// TIA Portal project "ElectricShipPLC" (V17)

(* hardware
DEVICE "S7-1200 station_2"  S7-1200 Station
   slot 0: "Rack_0"  S7-1200 Rack  Rack  V1.0
   slot 1: "PLC_3"  CPU 1214C DC/DC/DC  6ES7 214-1AG40-0XB0  V4.5
*)

// ===== PLC "PLC_3"  CPU 1214C DC/DC/DC =====

TYPE "TypeTx"
   STRUCT
      Droopout1 : LReal;
      Droopout2 : LReal;
      Breakerout1 : LReal;
      Breakerout2 : LReal;
      Breakerout3 : LReal;
   END_STRUCT;
END_TYPE

TYPE "TypeRx"
   STRUCT
      Droop1 : LReal;
      Droop2 : LReal;
      Breaker1 : LReal;
      Breaker2 : LReal;
      Breaker3 : LReal;
      Breaker4 : LReal;
   END_STRUCT;
END_TYPE

DATA_BLOCK "ModbusClientTx30_DB"   // DB5
{ S7_Optimized_Access := 'FALSE' }
VERSION : 0.1
// stored: InstanceOfName ModbusClientTx30
"ModbusClientTx30"
BEGIN
END_DATA_BLOCK

DATA_BLOCK "ModbusClientRx30_DB"   // DB7
{ S7_Optimized_Access := 'FALSE' }
VERSION : 0.1
// stored: InstanceOfName ModbusClientRx30
"ModbusClientRx30"
BEGIN
END_DATA_BLOCK

DATA_BLOCK "ModbusData"   // DB100
{ S7_Optimized_Access := 'TRUE' }
VERSION : 0.1
   VAR
      connectParamTx30 : TCON_IP_v4;
      connectParamRx30 : TCON_IP_v4;
      DataTx30 : Struct
         request : Bool := true;
         disconnect : Bool;
         done : Bool;
         busy : Bool;
         error : Bool;
         status : Word;
         statusSave : Word;
         modbusMode : USInt := 116;
         modbusDataAddress : UDInt := 0;
         modbusDataLen : UInt := 20;
      END_STRUCT;
      DataRx30 : Struct
         request : Bool := true;
         disconnect : Bool;
         done : Bool;
         busy : Bool;
         error : Bool;
         status : Word;
         statusSave : Word;
         modbusMode : USInt := 103;
         modbusDataAddress : UDInt := 20;
         modbusDataLen : UInt := 24;
      END_STRUCT;
      RegistersTx30Raw : Array[0..19] of Word;
      RegistersRx30Raw : Array[0..23] of Word;
      RegistersTx30 : "TypeTx";
      RegistersRx30 : "TypeRx";
   END_VAR
BEGIN
   connectParamTx30.LocalPort := 0;
   connectParamTx30.RemotePort := 502;
   connectParamTx30.RemoteAddress.ADDR[4] := 30;
   connectParamTx30.RemoteAddress.ADDR[3] := 0;
   connectParamTx30.RemoteAddress.ADDR[2] := 168;
   connectParamTx30.RemoteAddress.ADDR[1] := 192;
   connectParamTx30.ActiveEstablished := 1;
   connectParamTx30.ConnectionType := 11;
   connectParamTx30.ID := 1;
   connectParamTx30.InterfaceId := 64;
   connectParamRx30.InterfaceId := 64;
   connectParamRx30.ID := 2;
   connectParamRx30.ConnectionType := 11;
   connectParamRx30.ActiveEstablished := 1;
   connectParamRx30.RemoteAddress.ADDR[1] := 192;
   connectParamRx30.RemoteAddress.ADDR[2] := 168;
   connectParamRx30.RemoteAddress.ADDR[3] := 0;
   connectParamRx30.RemoteAddress.ADDR[4] := 30;
   connectParamRx30.RemotePort := 502;
   connectParamRx30.LocalPort := 0;
   RegistersTx30.Breakerout3 := 50.0;
   RegistersTx30.Breakerout1 := 10.0;
   RegistersTx30.Droopout2 := 10.0;
   RegistersTx30.Droopout1 := 100.0;
END_DATA_BLOCK

FUNCTION_BLOCK "ModbusClientRx30"   // FB2, SCL
{ S7_Optimized_Access := 'FALSE' }
VERSION : 0.1
   VAR_INPUT
      request : Bool;
      disconnect : Bool;
      modbusMode : USInt;
      modbusDataAddress : UDInt;
      modbusDataLen : UInt;
   END_VAR
   VAR_OUTPUT
      done : Bool;
      busy : Bool;
      error : Bool;
      status : Word;
   END_VAR
   VAR_IN_OUT
      connectParamClient : Variant;
      dataBuffer : Variant;
   END_VAR
   VAR
      instModbusClient : MB_CLIENT;
   END_VAR
BEGIN
   #instModbusClient(REQ:=#request,
                     DISCONNECT:=#disconnect,
                     MB_MODE:=#modbusMode,
                     MB_DATA_ADDR:=#modbusDataAddress,
                     MB_DATA_LEN:=#modbusDataLen,
                     DONE=>#done,
                     BUSY=>#busy,
                     ERROR=>#error,
                     STATUS=>#status,
                     MB_DATA_PTR:=#dataBuffer,
                     CONNECT:=#connectParamClient);
END_FUNCTION_BLOCK

FUNCTION_BLOCK "ModbusClientTx30"   // FB5, SCL
{ S7_Optimized_Access := 'FALSE' }
VERSION : 0.1
   VAR_INPUT
      request : Bool;
      disconnect : Bool;
      modbusMode : USInt;
      modbusDataAddress : UDInt;
      modbusDataLen : UInt;
   END_VAR
   VAR_OUTPUT
      done : Bool;
      busy : Bool;
      error : Bool;
      status : Word;
   END_VAR
   VAR_IN_OUT
      connectParamClient : Variant;
      dataBuffer : Variant;
   END_VAR
   VAR
      instModbusClient : MB_CLIENT;
   END_VAR
BEGIN
   #instModbusClient(REQ:=#request,
                     DISCONNECT:=#disconnect,
                     MB_MODE:=#modbusMode,
                     MB_DATA_ADDR:=#modbusDataAddress,
                     MB_DATA_LEN:=#modbusDataLen,
                     DONE=>#done,
                     BUSY=>#busy,
                     ERROR=>#error,
                     STATUS=>#status,
                     MB_DATA_PTR:=#dataBuffer,
                     CONNECT:=#connectParamClient);
END_FUNCTION_BLOCK

FUNCTION "Copy_Variant" : Void   // FC1, SCL
{ S7_Optimized_Access := 'FALSE' }
VERSION : 0.1
   VAR_IN_OUT
      source : Variant;
      destination : Variant;
   END_VAR
   VAR_TEMP
      tempStore : Array[0..199] of Byte;
      tempPos : DInt;
      tempRetval : Int;
   END_VAR
BEGIN
   #tempPos := 0;
   #tempRetval := Serialize(SRC_VARIABLE := #source,
                            DEST_ARRAY => #tempStore,
                            POS := #tempPos);

   #tempPos := 0;
   #tempRetval := Deserialize(SRC_ARRAY := #tempStore,
                              DEST_VARIABLE => #destination,
                              POS := #tempPos);
END_FUNCTION

ORGANIZATION_BLOCK "Main"   // OB1, LAD, ProgramCycle
TITLE = "Main Program Sweep (Cycle)"
{ S7_Optimized_Access := 'TRUE' }
VERSION : 0.1
   VAR_INPUT
      Initial_Call : Bool;   // Initial call of this OB
      Remanence : Bool;   // =True, if remanent data are available
   END_VAR
BEGIN
END_ORGANIZATION_BLOCK

ORGANIZATION_BLOCK "Cyclic interrupt"   // OB30, SCL, CyclicInterrupt
{ S7_Optimized_Access := 'TRUE' }
VERSION : 0.1
   VAR_INPUT
      Initial_Call : Bool;   // Initial call of this OB
      Event_Count : Int;   // Events discarded
   END_VAR
   VAR_TEMP
      ret : DWord;
      tempPos : DInt;
      tempRetval : Int;
   END_VAR
BEGIN
   // Read holding registers of server 30
   "ModbusClientRx30_DB"(request := "ModbusData".DataRx30.request,
                         disconnect := "ModbusData".DataRx30.disconnect,
                         modbusMode := "ModbusData".DataRx30.modbusMode,
                         modbusDataAddress := "ModbusData".DataRx30.modbusDataAddress,
                         modbusDataLen := "ModbusData".DataRx30.modbusDataLen,
                         done => "ModbusData".DataRx30.done,
                         busy => "ModbusData".DataRx30.busy,
                         error => "ModbusData".DataRx30.error,
                         status => "ModbusData".DataRx30.status,
                         connectParamClient := "ModbusData".connectParamRx30,
                         dataBuffer := "ModbusData".RegistersRx30Raw);
   IF "ModbusData".DataRx30.error <> 0 THEN
       "ModbusData".DataRx30.statusSave := "ModbusData".DataRx30.status;
   ELSE
       "Copy_Variant"(source := "ModbusData".RegistersRx30Raw,
                      destination := "ModbusData".RegistersRx30);
   END_IF;

   "ModbusData".RegistersTx30.Droopout1 := "ModbusData".RegistersRx30.Droop1;
   "ModbusData".RegistersTx30.Droopout2 := "ModbusData".RegistersRx30.Droop2;
   "ModbusData".RegistersTx30.Breakerout1 := "ModbusData".RegistersRx30.Breaker1;
   "ModbusData".RegistersTx30.Breakerout2 := "ModbusData".RegistersRx30.Breaker2;
   "ModbusData".RegistersTx30.Breakerout3 := "ModbusData".RegistersRx30.Breaker3;

   // Write holding registers of server 30
   "Copy_Variant"(source := "ModbusData".RegistersTx30,
                  destination := "ModbusData".RegistersTx30Raw);
   "ModbusClientTx30_DB"(request := "ModbusData".DataTx30.request,
                         disconnect := "ModbusData".DataTx30.disconnect,
                         modbusMode := "ModbusData".DataTx30.modbusMode,
                         modbusDataAddress := "ModbusData".DataTx30.modbusDataAddress,
                         modbusDataLen := "ModbusData".DataTx30.modbusDataLen,
                         done => "ModbusData".DataTx30.done,
                         busy => "ModbusData".DataTx30.busy,
                         error => "ModbusData".DataTx30.error,
                         status => "ModbusData".DataTx30.status,
                         connectParamClient := "ModbusData".connectParamTx30,
                         dataBuffer := "ModbusData".RegistersTx30Raw);
   IF "ModbusData".DataTx30.error <> 0 THEN
       "ModbusData".DataTx30.statusSave := "ModbusData".DataTx30.status;
   END_IF;
END_ORGANIZATION_BLOCK